FUNCTION_BLOCK Motor_Status (* Composite Function Block Type *)
  (* Standard: 61499-2 *)
  (* Version 0.0, 2/5/2026, Schneider Electric, template *)
  PACKAGE Hidryco.HidrycoLib;
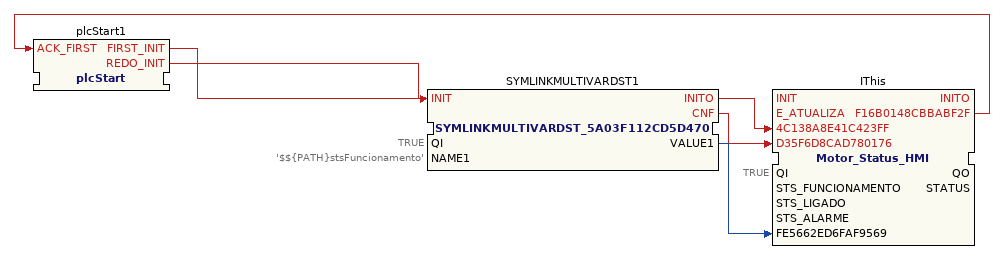
  FBS
    IThis : Motor_Status_HMI(QI := TRUE);
    SYMLINKMULTIVARDST1 : SYMLINKMULTIVARDST_5A03F112CD5D470(QI := TRUE, NAME1 := '$${PATH}stsFuncionamento'); {SET_ATTRIBUTE(Configuration.GenericFBType.InterfaceParams, Runtime.System#I:=1;VALUE${I$}:INT)}
    plcStart1 : plcStart;
  END_FBS
  EVENT_CONNECTIONS
    IThis.F16B0148CBBABF2F TO plcStart1.ACK_FIRST;
    plcStart1.FIRST_INIT TO SYMLINKMULTIVARDST1.INIT;
    plcStart1.REDO_INIT TO SYMLINKMULTIVARDST1.INIT;
    SYMLINKMULTIVARDST1.INITO TO IThis.4C138A8E41C423FF;
    SYMLINKMULTIVARDST1.CNF TO IThis.D35F6D8CAD780176;
  END_CONNECTIONS
  DATA_CONNECTIONS
    SYMLINKMULTIVARDST1.VALUE1 TO IThis.FE5662ED6FAF9569;
  END_CONNECTIONS
END_FUNCTION_BLOCK
